{attribute 'qualified_only'}
{attribute 'strict'}
TYPE E_ReworkDataState :
(
	Undefined := 0,
	CheckRequest,
	UpdateReworkData,
	Done,
	Error
);
END_TYPE

(* stored: Version 1.1.0.1, ProductVersion 3.1.4024.5
   DUT E_ReworkDataState: Id {ce1c2c31-fa59-4f18-8e5e-f5a7b98b2864} *)
